FUNCTION_BLOCK C_RESTART_CLIENT (* Composite Function Block Type *)
  (* Standard: 61499-2 *)
  (* Version 0.0, 2016-02-15, 4DIAC-IDE, 4DIAC-Consortium *)
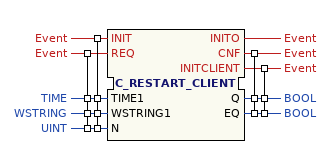
  EVENT_INPUT
    INIT WITH TIME1, WSTRING1, N;
    REQ WITH TIME1, WSTRING1, N; (* Normal Execution Request *)
  END_EVENT
  EVENT_OUTPUT
    INITO;
    CNF WITH Q, EQ; (* Execution Confirmation *)
    INITCLIENT WITH Q, EQ;
  END_EVENT
  VAR_INPUT
    TIME1 : TIME; (* time between each try of intializate and terminate the communication FB *)
    WSTRING1 : WSTRING; (* STATUS_CLIENT *)
    N : UINT; (* Number of tries(1-999),(0=infinite number of tries) *)
  END_VAR
  VAR_OUTPUT
    Q : BOOL; (* QI_CLIENT *)
    EQ : BOOL; (* (STATUS_CLIENT=="OK")=EQ *)
  END_VAR
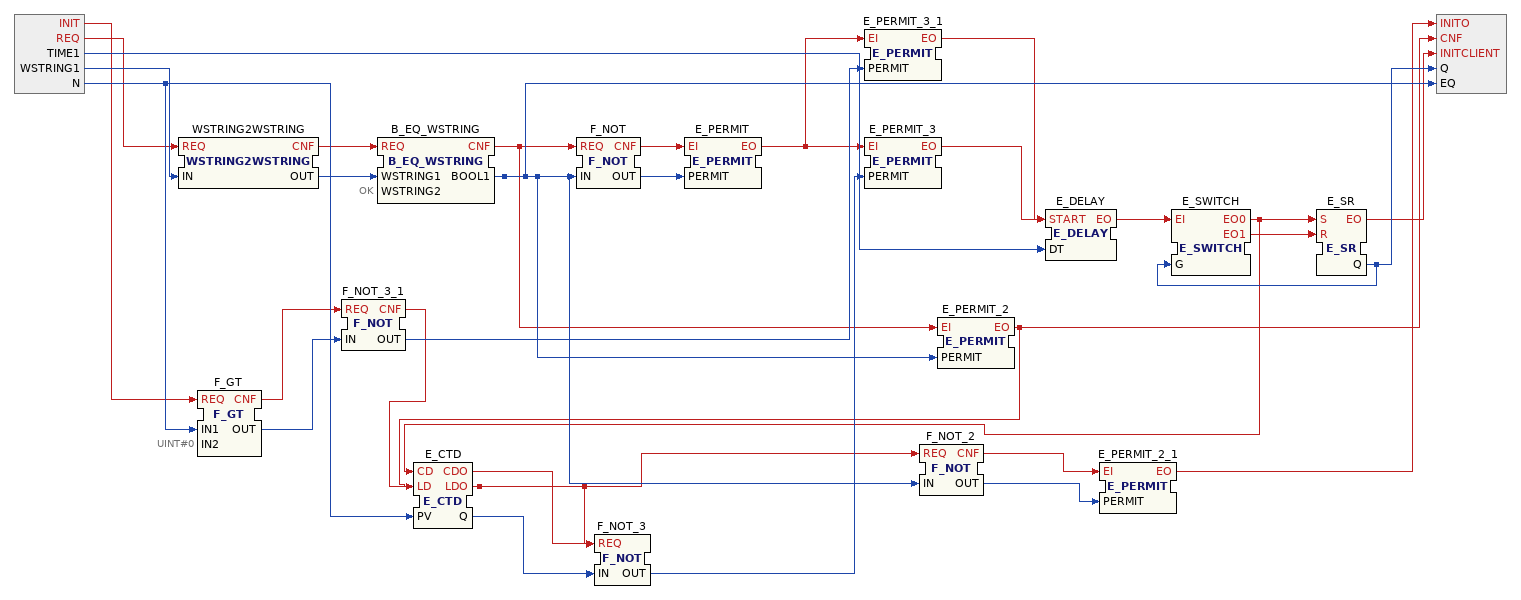
  FBS
    WSTRING2WSTRING : WSTRING2WSTRING;
    B_EQ_WSTRING : B_EQ_WSTRING(WSTRING2 := OK);
    E_DELAY : E_DELAY;
    E_SR : E_SR;
    E_SWITCH : E_SWITCH;
    E_PERMIT : E_PERMIT;
    F_NOT : F_NOT;
    E_PERMIT_2 : E_PERMIT;
    E_PERMIT_3 : E_PERMIT;
    E_CTD : E_CTD;
    F_NOT_3 : F_NOT;
    F_GT : F_GT(IN2 := UINT#0);
    E_PERMIT_3_1 : E_PERMIT;
    F_NOT_3_1 : F_NOT;
    E_PERMIT_2_1 : E_PERMIT;
    F_NOT_2 : F_NOT;
  END_FBS
  EVENT_CONNECTIONS
    WSTRING2WSTRING.CNF TO B_EQ_WSTRING.REQ;
    F_NOT.CNF TO E_PERMIT.EI;
    B_EQ_WSTRING.CNF TO F_NOT.REQ;
    E_SWITCH.EO0 TO E_SR.S;
    E_SWITCH.EO1 TO E_SR.R;
    E_DELAY.EO TO E_SWITCH.EI;
    E_SR.EO TO INITCLIENT;
    E_PERMIT_2.EO TO CNF;
    B_EQ_WSTRING.CNF TO E_PERMIT_2.EI;
    E_PERMIT_3.EO TO E_DELAY.START;
    E_PERMIT.EO TO E_PERMIT_3.EI;
    E_CTD.CDO TO F_NOT_3.REQ;
    E_SWITCH.EO0 TO E_CTD.CD;
    E_CTD.LDO TO F_NOT_3.REQ;
    REQ TO WSTRING2WSTRING.REQ;
    INIT TO F_GT.REQ;
    E_PERMIT.EO TO E_PERMIT_3_1.EI;
    E_PERMIT_3_1.EO TO E_DELAY.START;
    F_GT.CNF TO F_NOT_3_1.REQ;
    F_NOT_3_1.CNF TO E_CTD.LD;
    E_PERMIT_2_1.EO TO INITO;
    E_PERMIT_2.EO TO E_CTD.LD;
    E_CTD.LDO TO F_NOT_2.REQ;
    F_NOT_2.CNF TO E_PERMIT_2_1.EI;
  END_CONNECTIONS
  DATA_CONNECTIONS
    WSTRING2WSTRING.OUT TO B_EQ_WSTRING.WSTRING1;
    WSTRING1 TO WSTRING2WSTRING.IN;
    F_NOT.OUT TO E_PERMIT.PERMIT;
    B_EQ_WSTRING.BOOL1 TO F_NOT.IN;
    TIME1 TO E_DELAY.DT;
    E_SR.Q TO E_SWITCH.G;
    E_SR.Q TO Q;
    B_EQ_WSTRING.BOOL1 TO EQ;
    B_EQ_WSTRING.BOOL1 TO E_PERMIT_2.PERMIT;
    N TO E_CTD.PV;
    E_CTD.Q TO F_NOT_3.IN;
    F_NOT_3.OUT TO E_PERMIT_3.PERMIT;
    N TO F_GT.IN1;
    F_GT.OUT TO F_NOT_3_1.IN;
    F_NOT_3_1.OUT TO E_PERMIT_3_1.PERMIT;
    F_NOT_2.OUT TO E_PERMIT_2_1.PERMIT;
    B_EQ_WSTRING.BOOL1 TO F_NOT_2.IN;
  END_CONNECTIONS
END_FUNCTION_BLOCK
